// TIA Portal V19 export
FUNCTION_BLOCK "FB_FW_Auftrag"   // FB9, LAD
{ S7_Optimized_Access := 'TRUE' }
// stored: AutoNumber false, MemoryReserve 100, SetENOAutomatically false
   VAR
      StepNbr : Int;
      Quelle : Int;
      Ziel : Int;
      Positionen { S7_SetPoint := 'True'} : Array[1..30] of "UDT_Auftrag_Pos";
      Frg_Einfahrt { S7_SetPoint := 'True'} : Bool;
      Frg_Ausfahrt : Bool;
      Frg_Ablauf : Bool;
   END_VAR
   VAR_TEMP
      pos : Int;
      setPoint : DInt;
      WT_DB : DB_ANY;
      nextStep : Bool;
      startStep : Bool;
      parkStep : Bool;
      befehlOk : Bool;
   END_VAR
   VAR CONSTANT
      Fahrzeit : DInt := 40;
   END_VAR
BEGIN

REGION Network 1 (SCL)
   IF NOT "DI_FW_1".ZST.BEREIT OR "DI_FW_1".ZST.FEHLER OR NOT "DI_FW_1".ZST.Auto OR NOT "DI_FW_1".ZST.Unten_li OR NOT "DI_FW_1".ZST.Unten_re THEN
       RETURN;
   END_IF;
END_REGION

REGION Network 2 (SCL): Initialisierung der Werte
   FOR #pos := 1 TO 30 DO
       #Positionen[#pos].Abholbar := "DB_POS".POS[#pos].belegt AND ("DB_POS".POS[#pos].Vorruf OR "DB_POS".POS[#pos].fertig) AND NOT "DB_POS".POS[#pos].Sperre_out AND NOT "DB_POS".POS[#pos].notFG_out;
       #Positionen[#pos].Fertig := #Positionen[#pos].Abholbar AND ("DB_POS".POS[#pos].Restzeit <= #Fahrzeit);
       #Positionen[#pos].Sperre := "DB_POS".POS[#pos].belegt OR "DB_POS".POS[#pos].Sperre_in OR "DB_POS".POS[#pos].notFG_in;

       #Positionen[#pos].CheckSperre := TRUE;

       IF #Positionen[#pos].Abholbar THEN
           #setPoint := "DB_POS".POS[#pos].Soll_Expozeit;
           IF #setPoint = 0 THEN
               #setPoint := 1;
           END_IF;

           #Positionen[#pos].Oldest := DINT_TO_REAL("DB_POS".POS[#pos].Verweilzeit) / DINT_TO_REAL(#setPoint);
       ELSE
           #Positionen[#pos].Oldest := 0;
       END_IF;

       IF "DB_POS".POS[#pos].next_WT > 0 THEN
           #WT_DB := UINT_TO_DB_ANY("DB_POS".POS[#pos].next_WT + 100);
           #Positionen[#pos].Wt_Typ := #WT_DB.;
           #Positionen[#pos].Wt_Cmd := #WT_DB.;
           #Positionen[#pos].WT_151 := #WT_DB.;
       ELSE
           #Positionen[#pos].Wt_Typ := 0;
           #Positionen[#pos].Wt_Cmd := 0;
           #Positionen[#pos].WT_151 := FALSE;
       END_IF;
   END_FOR;
END_REGION

REGION Network 3 (SCL)
   CASE #StepNbr OF
       1:  // Schritt 1 CM01/CMD02 -> CM03
           IF "DB_ANLAGE".config.NormalB THEN
               "FC_FW_Auftrag_Step1_NB"(Frg_Schritt := #Frg_Ablauf,
                                        nextStep => #nextStep,
                                        startStep => #startStep,
                                        parkStep => #parkStep,
                                        Quelle := #Quelle,
                                        Ziel := #Ziel,
                                        Positionen := #Positionen);
           ELSE
               "FC_FW_Auftrag_Step1_KB"(Frg_Schritt := #Frg_Ablauf,
                                        nextStep => #nextStep,
                                        startStep => #startStep,
                                        parkStep => #parkStep,
                                        Quelle := #Quelle,
                                        Ziel := #Ziel,
                                        Positionen := #Positionen);
           END_IF;

       2:        // Schritt 1 CM03 -> CM01/CM02
           IF "DB_ANLAGE".config.NormalB THEN
               "FC_FW_Auftrag_Step2_NB"(Frg_Schritt := #Frg_Ablauf,
                                        nextStep => #nextStep,
                                        startStep => #startStep,
                                        parkStep => #parkStep,
                                        Quelle := #Quelle,
                                        Ziel := #Ziel,
                                        Positionen := #Positionen);
           ELSE
               "FC_FW_Auftrag_Step2_KB"(Frg_Schritt := #Frg_Ablauf,
                                        nextStep => #nextStep,
                                        startStep => #startStep,
                                        parkStep => #parkStep,
                                        Quelle := #Quelle,
                                        Ziel := #Ziel,
                                        Positionen := #Positionen);
           END_IF;

       3:  // Schritt 3 CM03 -> CM04
           IF "DB_ANLAGE".config.NormalB THEN
               "FC_FW_Auftrag_Step3_NB"(Frg_Schritt := #Frg_Ablauf,
                                        nextStep => #nextStep,
                                        startStep => #startStep,
                                        parkStep => #parkStep,
                                        Quelle := #Quelle,
                                        Ziel := #Ziel,
                                        Positionen := #Positionen);
           ELSE
               "FC_FW_Auftrag_Step3_KB"(Frg_Schritt := #Frg_Ablauf,
                                        nextStep => #nextStep,
                                        startStep => #startStep,
                                        parkStep => #parkStep,
                                        Quelle := #Quelle,
                                        Ziel := #Ziel,
                                        Positionen := #Positionen);
           END_IF;

       4:  // Schritt 4 WR02 -> CM03
           IF "DB_ANLAGE".config.NormalB THEN
               "FC_FW_Auftrag_Step4_NB"(Frg_Einfahrt := #Frg_Einfahrt,
                                        Frg_Schritt := #Frg_Ablauf,
                                        nextStep => #nextStep,
                                        startStep => #startStep,
                                        parkStep => #parkStep,
                                        Quelle := #Quelle,
                                        Ziel := #Ziel,
                                        Positionen := #Positionen);
           ELSE
               "FC_FW_Auftrag_Step4_KB"(Frg_Einfahrt := #Frg_Einfahrt,
                                        Frg_Schritt := #Frg_Ablauf,
                                        nextStep => #nextStep,
                                        startStep => #startStep,
                                        parkStep => #parkStep,
                                        Quelle := #Quelle,
                                        Ziel := #Ziel,
                                        Positionen := #Positionen);
           END_IF;

       5:  // Schritt 5 CM04 -> WR02
           IF  "DB_ANLAGE".config.NormalB THEN
               "FC_FW_Auftrag_Step5_NB"(Frg_Schritt := #Frg_Ablauf,
                                        nextStep => #nextStep,
                                        startStep => #startStep,
                                        parkStep => #parkStep,
                                        Quelle := #Quelle,
                                        Ziel := #Ziel,
                                        Positionen := #Positionen,
                                        Frg_Ausfahrt := #Frg_Ausfahrt);
           ELSE
               "FC_FW_Auftrag_Step5_KB"(Frg_Schritt := #Frg_Ablauf,
                                        nextStep => #nextStep,
                                        startStep => #startStep,
                                        parkStep => #parkStep,
                                        Quelle := #Quelle,
                                        Ziel := #Ziel,
                                        Positionen := #Positionen,
                                        Frg_Ausfahrt := #Frg_Ausfahrt);
           END_IF;

       6:  //Parken
           "FC_FW_Auftrag_Parken"(nextStep => #nextStep,
                                  startStep=>#startStep,
                                  Quelle := #Quelle,
                                  Ziel := #Ziel,
                                  Positionen := #Positionen);

       ELSE  // Initialisieren
           #nextStep := FALSE;
           #startStep := TRUE;
           #parkStep := FALSE;
   END_CASE;

   IF #startStep THEN
       //von vorn beginnen
       #StepNbr := 1;
   ELSIF #nextStep THEN
       //weiterschalten
       #StepNbr := #StepNbr + 1;
   ELSIF #parkStep THEN
       //parken
       #StepNbr := 6;
   ELSE
       //warten
       ;
   END_IF;
END_REGION
END_FUNCTION_BLOCK
